// TIA Portal V20 export
DATA_BLOCK "Instance_FB_Visual_Test_DB"   // DB107
// stored: AutoNumber false, InstanceOfName FB_Visual_Test, InstanceOfType FB
"FB_Visual_Test"
   // VAR_INPUT
   //    Star_Functional_Test : Bool;
   //    Reset_Functional_Test : Bool;
   //    Button_Start_Approve : Bool;
   //    In_Test_Parameters : "IO_Device_Test_Parameters";
   // END_VAR
   // VAR_OUTPUT
   //    Visual_Test_Approved_PLC : Bool;
   // END_VAR
   // VAR
   //    Aux_Trigger : Bool;
   //    Timer_Delay_Start_Visual_Test { S7_SetPoint := 'True'} : TON_TIME;
   //    Timer_Delay_Reset { S7_SetPoint := 'True'} : TON_TIME;
   // END_VAR
BEGIN
END_DATA_BLOCK
